FUNCTION_BLOCK DrillStation_FBDKTestBench (* Composite Function Block Type *)
  (* Standard: 61499-2 *)
  (* Version 0.2, 2003-12-05, JHC, Rockwell Automation, Renamed from NEWCOMPFB. *)
  (* Version 0.1, 2002-01-08, JHC, Rockwell Automation, Added DLY FB as example. *)
  (* Version 0.0, 2000-05-27, JHC, Rockwell Automation *)
  (* Compiler header: package fb.rt.benchmarks.DrillStation; *)
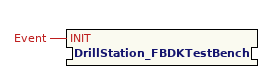
  EVENT_INPUT
    INIT; (* Initialization Request *)
  END_EVENT
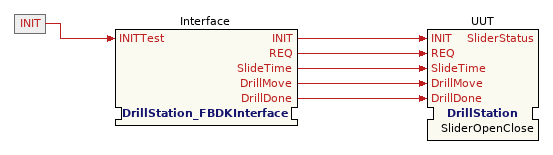
  FBS
    Interface : DrillStation_FBDKInterface;
    UUT : DrillStation;
  END_FBS
  EVENT_CONNECTIONS
    INIT TO Interface.INITTest;
    Interface.INIT TO UUT.INIT;
    Interface.REQ TO UUT.REQ;
    Interface.SlideTime TO UUT.SlideTime;
    Interface.DrillMove TO UUT.DrillMove;
    Interface.DrillDone TO UUT.DrillDone;
  END_CONNECTIONS
END_FUNCTION_BLOCK
